SUBAPPLICATION Fahrwerk_Mittelpunkt_Anzeige (* Reine Anzeige-Haelfte von Fahrwerk_Mittelpunkt_Automatik, herausgeloest: 2 Bargraphen + Status-Center-Hintergrundfarbe fuer einen Winkelsensor mit Mittelstellung (Achslenkung/Hangausgleich), gespeist von einem lokal bereits verfuegbaren AR-Plug (CAL_IN) statt einem eigenen OPC-UA-Self-Subscribe. Fuer Faelle, in denen die eigentliche Automatik (AUTO_LINKS/RECHTS-Regelung) auf einer anderen Station laeuft als die VT (z.B. Hangausgleich seit dem Umzug nach STG4), dort aber trotzdem eine Anzeige gebraucht wird - Franz: 'Bargraph braucht es. Wobei die Frage ist ob das ein extra forwarding sein muss? Fuer die CAL Maske bei Eingaenge brauchen wir den kalibrierten Wert ohnehin schon.' Kein extra Forwarding noetig: der Kalibrierkanal-Konsument (logiBUS_AI_Calibrated_Subscribe_VT_(3P_)OPC) hat den Wert bereits lokal als CAL_OUT-Plug, genau der wird hier direkt weiterverdrahtet. *)
  (* Standard: 61499-2; Description: Copyright (c) 2026 Meisterschulen am Ostbahnhof This program and the accompanying materials are made available under the terms of the Eclipse Public License 2.0 which is available at https://www.eclipse.org/legal/epl-2.0/ SPDX-License-Identifier: EPL-2.0 *)
  (* Version 1.0, 2026-09-26, Franz Höpfinger, Meisterschulen am Ostbahnhof, initial implementation - herausgeloest aus Fahrwerk_Mittelpunkt_Automatik.SUB (SUBSCRIBE_Y/SPLIT_Y/CENTER_CMP/SplitBar/STATUS_CENTER_BG kamen dort bereits genauso vor), fuer Hangausgleich: die Automatik selbst laeuft seit v3.0 auf STG4 (kein VT dort, u16ObjId_Status_Center/stObjBargraphSplit dort bewusst ID_NULL), diese SubApp laeuft stattdessen auf STG1, gespeist vom ohnehin schon lokal vorhandenen CAL_OUT-Plug der Kalibrierkanal-Konsumenten-Instanz - kein zusaetzlicher Remote-Round-Trip. *)
  PACKAGE MyLib::sys;
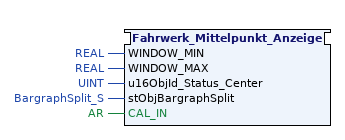
  VAR_INPUT
    WINDOW_MIN : REAL := -2.0; (* Untere Fenstergrenze (%), ab wann 'links ausgelenkt' gilt - muss zum WINDOW_MIN der zugehoerigen Fahrwerk_Mittelpunkt_Automatik-Instanz passen *)
    WINDOW_MAX : REAL := 2.0; (* Obere Fenstergrenze (%), ab wann 'rechts ausgelenkt' gilt - siehe WINDOW_MIN *)
    u16ObjId_Status_Center : UINT; (* Object ID Status_Center-Button (Achslenkung_Status_Center bzw. Hangausgleich_Status_Center, '><'-Indikator) *)
    stObjBargraphSplit : isobus::utils::bargraph::BargraphSplit_S; (* Object IDs der 2 Bargraphen + gemeinsame Betrags-Grenzen, siehe FBs::const::DefaultPool_BargraphSplit::Bargraph_Achslenkung_BargraphSplit bzw. _Hangausgleich_BargraphSplit *)
  END_VAR
  SOCKETS
    CAL_IN : adapter::types::unidirectional::AR; (* Kalibrierter Winkel von aussen (z.B. AnalogChannel_Hangausgleich_Winkel.CAL_OUT), statt eigenem lokalen OPC-UA-Self-Subscribe *)
  END_SOCKETS
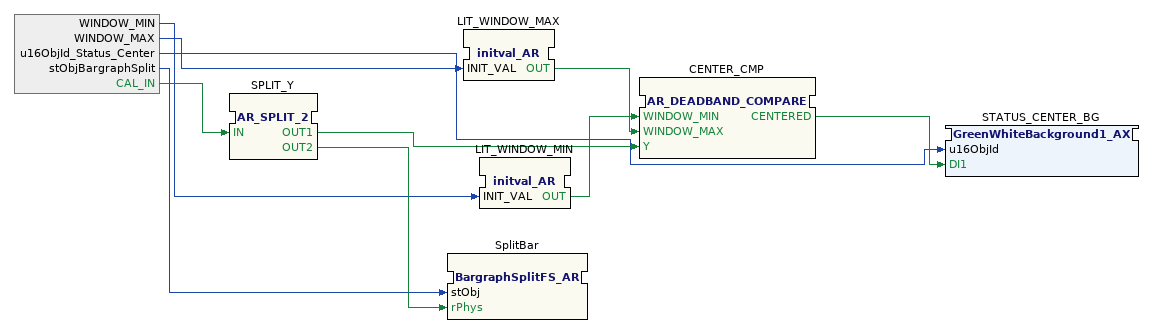
  FBS
    SPLIT_Y : adapter::events::unidirectional::AR_SPLIT_2;
    CENTER_CMP : adapter::Engineering::measurements::AR_DEADBAND_COMPARE;
    LIT_WINDOW_MIN : adapter::types::unidirectional::AR::initval::initval_AR;
    LIT_WINDOW_MAX : adapter::types::unidirectional::AR::initval::initval_AR;
    SplitBar : isobus::UT::Q::BargraphSplitFS_AR;
  END_FBS
  SUBAPPS
    STATUS_CENTER_BG : MyLib::sys::GreenWhiteBackground1_AX;
  END_SUBAPPS
  DATA_CONNECTIONS
    WINDOW_MIN TO LIT_WINDOW_MIN.INIT_VAL;
    WINDOW_MAX TO LIT_WINDOW_MAX.INIT_VAL;
    u16ObjId_Status_Center TO STATUS_CENTER_BG.u16ObjId;
    stObjBargraphSplit TO SplitBar.stObj;
  END_CONNECTIONS
  ADAPTER_CONNECTIONS
    CAL_IN TO SPLIT_Y.IN;
    LIT_WINDOW_MIN.OUT TO CENTER_CMP.WINDOW_MIN;
    LIT_WINDOW_MAX.OUT TO CENTER_CMP.WINDOW_MAX;
    SPLIT_Y.OUT1 TO CENTER_CMP.Y;
    SPLIT_Y.OUT2 TO SplitBar.rPhys;
    CENTER_CMP.CENTERED TO STATUS_CENTER_BG.DI1;
  END_CONNECTIONS
END_SUBAPPLICATION
